# B&R Automation Studio project PickNPlaceD5Demo (part 2)

#### DeviceActions.st
```iecst
ACTION updateProductData:

	FOR i:=0 TO MAX_TRACKING_FRAMES DO
		IF (Products[i].TrackingFrameID <> 0 AND Products[i].Attribute <> 0) THEN
			ProdDetails ACCESS Products[i].Attribute;
			brsmemcpy(ADR(ProdDetails.Pos), ADR(Products[i].CurrentPosition), SIZEOF(McPosType));
			ProdDetails.This := ADR(ProdDetails);
			ProdDetails.TrackingFrameID := Products[i].TrackingFrameID;
		END_IF
	END_FOR

END_ACTION

ACTION deleteOutOfScopeProducts:

	FOR i:=0 TO MAX_TRACKING_FRAMES DO
		IF Products[i].Distance >= ConvSettings.DeletePosition THEN // todo: distance as a constant!
			IF (Products[i].Attribute <> 0) THEN
				brsmemset(Products[i].Attribute, 0, SIZEOF(ProductDetailsType));
			END_IF
			MC_BR_TrackingFrameDelete_0.Mode := mcTRKFRM_DELETE_MOD_FRAME;
			MC_BR_TrackingFrameDelete_0.TrackingFrameID	:= Products[i].TrackingFrameID;
			MC_BR_TrackingFrameDelete_0.Execute	:= TRUE;
			EXIT;
		END_IF
	END_FOR

END_ACTION

ACTION addNewObjects:

	LastProductPosition := MpAxConveyor.Position;

	// Generate a random Y Position --> Here a vision sensor informatin is needed in real systems
	MC_BR_TrackingFrameCreate_0.Parameters.Translation.Y := ConvSettings.YShift;

	// Add attributes memory
	FOR i := 0 TO MAX_TRACKING_FRAMES DO
		IF ProductDetails[i].TrackingFrameID = 0 THEN
			brsmemset(ADR(ProductDetails[i]), 0, SIZEOF(ProductDetailsType));
			MC_BR_TrackingFrameCreate_0.Parameters.Attribute := ADR(ProductDetails[i]);
			EXIT;
		END_IF
	END_FOR

	// Add frame in the buffer
	MC_BR_TrackingFrameCreate_0.Parameters.LatchedPath.Position := LastProductPosition;
	MC_BR_TrackingFrameCreate_0.Execute	:= TRUE;

END_ACTION

ACTION updateSceneViewerPositions:

	FOR i:= 0 TO MAX_TRACKING_FRAMES DO
		ProductsPosition[i].Valid := Products[i].TrackingFrameID <> 0;

		IF Products[i].Attribute <> 0 THEN
			ProdDetails ACCESS Products[i].Attribute;
			IF ProdDetails.InTracking THEN
				ProductsPosition[i].Material := 4; //yellow
			ELSE
				ProductsPosition[i].Material := 1; //red
			END_IF
			ProductsPosition[i].Full := ProdDetails.Used;
			ProductsPosition[i].Empty := NOT ProdDetails.Used;
			ProductsPosition[i].Element1 := ProdDetails.Element1;
			ProductsPosition[i].Element2 := ProdDetails.Element2;
		ELSE
			ProductsPosition[i].Full := FALSE;
			ProductsPosition[i].Empty := FALSE;
			ProductsPosition[i].Element1 := FALSE;
			ProductsPosition[i].Element2 := FALSE;
			ProductsPosition[i].Material := 1;
		END_IF

		ProductsPosition[i].PositionX := LREAL_TO_REAL(Products[i].CurrentPosition.X);
		ProductsPosition[i].PositionY := LREAL_TO_REAL(Products[i].CurrentPosition.Y);
		ProductsPosition[i].PositionZ := LREAL_TO_REAL(Products[i].CurrentPosition.Z);
	END_FOR

END_ACTION

ACTION applyBeltMovement:

	IF AxWithCommandConsideration THEN
		IF NOT MC_MoveAdditive_0.Busy THEN
			MC_MoveAdditive_0.Distance := ConvSettings.IndexingDistance;
			MC_MoveAdditive_0.Velocity := ConvSettings.VelocityProduction;
			MC_MoveAdditive_0.BufferMode := mcABORTING;
			MC_MoveAdditive_0.Execute := TRUE;
		END_IF
	ELSE
		MC_MoveVelocity_0.Velocity := ConvSettings.VelocityProduction;
		MC_MoveVelocity_0.Execute := MC_MoveVelocity_0.InVelocity OR NOT MC_MoveVelocity_0.Busy;
	END_IF

END_ACTION

ACTION resetFUBs:

	IF (MpAxConveyor.Update AND MpAxConveyor.UpdateDone) OR MpAxConveyor.Error THEN
		MpAxConveyor.Update	:= FALSE;
	END_IF

	IF (NOT(MpAxConveyor.MoveActive) AND NOT(MpAxConveyor.CommandBusy)) OR MpAxConveyor.Error THEN
		MpAxConveyor.MoveVelocity := FALSE;
		MpAxConveyor.Update := FALSE;
	END_IF

	IF MpAxConveyor.ErrorReset AND NOT(MpAxConveyor.Error) THEN
		MpAxConveyor.ErrorReset := FALSE;
	END_IF

	IF (MpAxConveyor.Home AND MpAxConveyor.IsHomed) OR MpAxConveyor.Error THEN
		MpAxConveyor.Home := FALSE;
	END_IF

	IF MC_BR_TrackingFrameCreate_0.Done OR MC_BR_TrackingFrameCreate_0.Error THEN
		MC_BR_TrackingFrameCreate_0.Execute	:= FALSE;
	END_IF

	IF MC_BR_TrackingFrameDelete_0.Done OR MC_BR_TrackingFrameDelete_0.Error THEN
		MC_BR_TrackingFrameDelete_0.Execute := FALSE;
	END_IF

	IF MC_MoveVelocity_0.Error OR MC_MoveVelocity_0.CommandAborted OR MC_MoveVelocity_0.Busy THEN
		MC_MoveVelocity_0.Execute := FALSE;
	END_IF

	IF MC_MoveAdditive_0.Error OR MC_MoveAdditive_0.CommandAborted OR MC_MoveAdditive_0.Busy OR MC_MoveAdditive_0.Done THEN
		MC_MoveAdditive_0.Execute := FALSE;
	END_IF

	IF MC_Stop_0.Error OR MC_Stop_0.CommandAborted OR MC_Stop_0.Busy OR MC_Stop_0.Done THEN
		MC_MoveAdditive_0.Execute := FALSE;
	END_IF

	IF MC_BR_TrackingPathReset_0.Busy OR MC_BR_TrackingPathReset_0.Error OR MC_BR_TrackingPathReset_0.Done THEN
		MC_BR_TrackingPathReset_0.Execute := FALSE;
	END_IF

	IF MC_BR_TrackingPathReadInfo_0.Error THEN
		MC_BR_TrackingPathReadInfo_0.Enable := FALSE;
	END_IF

END_ACTION

ACTION initConveyor:

	// Configure Frame Buffer, to get actual pointer to Products --> Check state of Products
	MC_BR_TrackingPathGetFrames_0.Parameters.CoordSystem := mcACS;
	MC_BR_TrackingPathGetFrames_0.Parameters.DataAddress := ADR(Products);
	MC_BR_TrackingPathGetFrames_0.Parameters.GetMode	:= mcTRKPATH_GET_MOD_ALL_FRAMES;
	MC_BR_TrackingPathGetFrames_0.Parameters.InfoMode	:= mcTRKPATH_INFO_MOD_ALL;
	MC_BR_TrackingPathGetFrames_0.Parameters.NumberOfFrames := MAX_TRACKING_FRAMES;
	MC_BR_TrackingPathGetFrames_0.Parameters.TrackingFrameID := 0;

	// Set Default Parameters of the Tracking Frames
	MC_BR_TrackingFrameCreate_0.Parameters.Attribute	:= 0;
	MC_BR_TrackingFrameCreate_0.Parameters.Translation.X := 0.0;
	MC_BR_TrackingFrameCreate_0.Parameters.Translation.Y := 0.0;
	MC_BR_TrackingFrameCreate_0.Parameters.Translation.Z := 0.0;
	MC_BR_TrackingFrameCreate_0.Parameters.Orientation.Angle1 := 0.0;
	MC_BR_TrackingFrameCreate_0.Parameters.Orientation.Angle2 := 0.0;
	MC_BR_TrackingFrameCreate_0.Parameters.Orientation.Angle3 := 0.0;
	MC_BR_TrackingFrameCreate_0.Parameters.Orientation.Type := 0;

	MC_BR_TrackingPathReadStatus_0.Enable := TRUE;
	MC_BR_TrackingPathReadInfo_0.Enable := TRUE;

	// Configuration of movement command
	MC_MoveAdditive_0.Acceleration := 1000;
	MC_MoveAdditive_0.Deceleration := 1000;
	MC_MoveAdditive_0.Jerk := 10000;
	MC_MoveAdditive_0.BufferMode := mcABORTING;

	MC_MoveVelocity_0.Acceleration := 1000;
	MC_MoveVelocity_0.Deceleration := 1000;
	MC_MoveVelocity_0.Direction := mcDIR_POSITIVE;
	MC_MoveVelocity_0.BufferMode := mcABORTING;

	MC_Stop_0.Deceleration := 1000;
	MC_Stop_0.Jerk := 10000;

	// Belt Position of fixed tracking frame
	ParkPosition := 0;

END_ACTION
```

### Program Logical/Conveyor/APP_ConveyorOut (IEC)

#### Init.st
```iecst
PROGRAM _INIT

	TrackLinkConveyor := ADR(gTrackingPathConveyorOut);
	AxGroupLink := ADR(AxConveyorOut);
	ConvSettings ACCESS ADR(ControlPanel.Input.Conveyor2);
	AxWithCommandConsideration := TRUE;

	initConveyor;

END_PROGRAM
```

- Cyclic.st (reference to Logical/Conveyor/APP_ConveyorIn/Cyclic.st)

- DeviceActions.st (reference to Logical/Conveyor/APP_ConveyorIn/DeviceActions.st)

- Variables.var (reference to Logical/Conveyor/APP_ConveyorIn/Variables.var)

### Package Logical/Robots/Robot1 - Device: Scara

### Program Logical/Robots/Robot1/APP_Robot1

#### CommonVars.var
```iecst
(*
Link handling*)
VAR
	AxQ1 : UDINT; (*Memory to Q1*)
	AxQ2 : UDINT; (*Memory to Q2*)
	AxQ3 : UDINT; (*Memory to Q4*)
	AxQ4 : UDINT; (*Memory to Q4*)
	AxQ5 : UDINT; (*Memory to Q4*)
	TrackLinkConveyorOut : UDINT; (*Link to conveyor tracking path*)
	TrackLinkConveyorIn : UDINT; (*Link to conveyor tracking path*)
	MpDeltaName : STRING[250]; (*Name of axGroup to find position in object hierachy*)
	MpLinkDelta : UDINT; (*Link to delta*)
	ProgramLink : REFERENCE TO STRING[32]; (*Program name as string executed by the interpreter*)
END_VAR
(*
Robot Definition*)
VAR
	MC_BR_MoveProgram_X : MC_BR_MoveProgram;
	MC_BR_GroupPower_X : MC_BR_GroupPower;
	MC_GroupStop_X : MC_GroupStop;
	MC_GroupReset_X : MC_GroupReset;
	MC_BR_GroupHome_X : MC_BR_GroupHome_15; (*Group object to home axis group*)
	MC_BR_GroupReadInfo_X : MC_BR_GroupReadInfo;
	MC_GroupContinue_X : MC_GroupContinue; (*Continue Interpreter in case of a new tracking Object*)
	MC_BR_TrackingStatus_PathGen_X : MC_BR_TrackingStatus_PathGen; (*Tracking Path, read all objects on Path*)
	MC_BR_PathInfo_X : MC_BR_PathInfo;
	MC_GroupReadStatus_X : MC_GroupReadStatus; (*Group object to home axis group*)
	MC_BR_PauseWorkspaceMonitoring_X : MC_BR_PauseWorkspaceMonitoring;
	MC_GroupReadActualPosition_X : MC_GroupReadActualPosition_15; (*Group object to home axis group*)
END_VAR
(*
Variables used handling objects and reading informations about the robot*)
VAR
	MC_BR_TrackingPathGetFrames_In : MC_BR_TrackingPathGetFrames; (*Tracking Path, read all objects on Path*)
	MC_BR_TrackingPathReadStatus_In : MC_BR_TrackingPathReadStatus;
	MC_BR_TrackingPathGetFrames_Out : MC_BR_TrackingPathGetFrames; (*Tracking Path, read all objects on Path*)
	MC_BR_TrackingPathReadStatus_Out : MC_BR_TrackingPathReadStatus;
END_VAR
(*
Logic*)
VAR
	State : DeviceStatesListEnum; (*Statemachine*)
	i : INT; (*loop counter*)
	j : INT; (*loop counter*)
	XPosMax : LREAL; (*Figure out object with min distance to the robot*)
	FeedrateReduction : LREAL; (*Feedrate reduction calculated based on the distance*)
	Products_Out : ARRAY[0..MAX_TRACKING_FRAMES] OF McTrkFrmInfoType; (*List of all Frames*)
	Products_In : ARRAY[0..MAX_TRACKING_FRAMES] OF McTrkFrmInfoType; (*List of all Frames*)
END_VAR
(*
Scene Viewer*)
VAR
	ProdDetails : REFERENCE TO ProductDetailsType; (*Scene Viewer*)
	PickTrackingObjectDetails : REFERENCE TO ProductDetailsType; (*Scene Viewer*)
	PlaceTrackingObjectDetails : REFERENCE TO ProductDetailsType; (*Scene Viewer*)
	Grab1Closed : BOOL;
	Grab2Closed : BOOL;
END_VAR
(*
ST Var*)
VAR
	MinPlacePosX : LREAL := 0; (*ST Var - Maximum reachable x position*)
	MaxPlacePosX : LREAL := 0; (*ST Var - Maximum reachable x position*)
	MinPickPosX : LREAL := 0; (*ST Var - Maximum reachable x position*)
	MaxPickPosX : LREAL := 0; (*ST Var - Maximum reachable x position*)
	PlaceTrackingObject : UDINT; (*ST Var - ADR(ProductDetailsType)*)
	PickTrackingObject : UDINT; (*ST Var - ADR(ProductDetailsType)*)
	M8 : BOOL; (*ST Var*)
	M9 : BOOL; (*ST Var*)
	M16 : BOOL; (*ST Var*)
	M17 : BOOL; (*ST Var*)
	M20 : BOOL; (*ST Var*)
	M21 : BOOL; (*ST Var*)
END_VAR
(*
Monitorin Elements*)
VAR
	BasicMonitor : McPathGenMonElemBasicMonType; (*Monitor to get interpreter line*)
	IPMonitor : McProgIntIpMonitorType; (*Monitor to get interpreter line*)
END_VAR
```

#### Cyclic.st
```iecst
PROGRAM _CYCLIC

	CASE State OF

		/////////////////////////////////////////////////////////////////////////////
		STATE_WAIT:
		/////////////////////////////////////////////////////////////////////////////
			IF  ControlPanel.Input.Start THEN
				State := STATE_INIT;
			END_IF

		/////////////////////////////////////////////////////////////////////////////
		STATE_INIT:
			/////////////////////////////////////////////////////////////////////////////
			IF NOT (MC_BR_TrackingPathReadStatus_In.TrackingPathReady OR MC_BR_TrackingPathReadStatus_Out.TrackingPathReady) THEN
				/// Wait
			ELSIF MC_BR_GroupHome_X.Busy OR MC_GroupReset_X.Busy OR NOT MC_GroupReadStatus_X.Valid OR NOT MC_BR_GroupReadInfo_X.Valid THEN
				// wait
			ELSIF MC_GroupReadStatus_X.Error OR MC_BR_GroupHome_X.Error OR MC_BR_GroupPower_X.Error OR MC_BR_MoveProgram_X.Error OR MC_GroupReset_X.Error OR MC_BR_GroupReadInfo_X.Error THEN
				MC_GroupReset_X.Execute := TRUE;

			ELSIF NOT MC_BR_GroupReadInfo_X.PowerOn THEN
				MC_BR_GroupPower_X.Enable := TRUE;

			ELSIF NOT MC_BR_GroupReadInfo_X.IsHomed	THEN
				MC_BR_GroupHome_X.Execute := TRUE;

			ELSIF MC_GroupReadStatus_X.GroupStandby THEN
				PickTrackingObject := 0;
				PlaceTrackingObject := 0;
				brsmemset(ADR(Products_In), 0, SIZEOF(Products_In));
				brsmemset(ADR(Products_Out), 0, SIZEOF(Products_Out));
				MC_BR_MoveProgram_X.Name := ProgramLink;
				MC_BR_MoveProgram_X.Execute := TRUE;
				MC_BR_PauseWorkspaceMonitoring_X.Enable := FALSE;
				State := STATE_PRODUCTION;

			END_IF

		/////////////////////////////////////////////////////////////////////////////
		STATE_PRODUCTION:
		/////////////////////////////////////////////////////////////////////////////

			// ------------------------------------------------------------------------------------------------------------------------------------------------
			// Case Pick Frame: choose which frame is the next to pick which is not already grabbed and not already in manipulation
			// ------------------------------------------------------------------------------------------------------------------------------------------------
			chooseNextSlots;

			// ------------------------------------------------------------------------------------------------------------------------------------------------
			// Case Grip Product: Hande M Commands on Tracked object
			// ------------------------------------------------------------------------------------------------------------------------------------------------
			handleMFunctions;

			// ------------------------------------------------------------------------------------------------------------------------------------------------
			// Case Scene Viewer Update Robot 1: Update Positions in Tracking case, to get a Scene Viewer Visu
			// ------------------------------------------------------------------------------------------------------------------------------------------------

			updateSceneViewer;

			// ------------------------------------------------------------------------------------------------------------------------------------------------
			// Case State M. Production : Handle End of Process
			// ------------------------------------------------------------------------------------------------------------------------------------------------
			IF MC_GroupReadStatus_X.Error OR MC_GroupReadStatus_X.GroupErrorStop OR MC_BR_MoveProgram_X.Error THEN
				State := STATE_ERROR;
				MC_GroupStop_X.Execute := TRUE;
				ControlPanel.Input.Start := FALSE;

			ELSIF NOT(ControlPanel.Input.Start) THEN

				MC_GroupStop_X.Execute := TRUE;
				MC_BR_GroupPower_X.Enable := FALSE;

				IF MC_GroupReadStatus_X.GroupDisabled THEN
					State := STATE_WAIT;

				ELSIF MC_GroupReadStatus_X.GroupErrorStop THEN
					State := STATE_ERROR;
				END_IF

			END_IF

		///////////////////////////////////////////////////////////////////////////////
		STATE_ERROR:
		///////////////////////////////////////////////////////////////////////////////
			IF MC_GroupReset_X.Busy OR MC_GroupReadStatus_X.Error OR MC_GroupReadStatus_X.GroupErrorStop THEN
				IF ControlPanel.Input.Reset THEN
					MC_GroupReset_X.Execute := NOT MC_GroupReset_X.Busy;
					MC_BR_GroupHome_X.Execute := NOT MC_BR_GroupHome_X.Busy;
				END_IF
			ELSE
				State := STATE_WAIT;
			END_IF

	END_CASE

	PlaceTrackingObjectDetails ACCESS PlaceTrackingObject;
	PickTrackingObjectDetails ACCESS PickTrackingObject;
	runFUBs;

END_PROGRAM
```

#### DefineLinks.st
```iecst
ACTION DefineLinks:

	// Define Links to the axes of the Robot
	AxQ1 := ADR(gAxisQ1_D5r1100R_1);
	AxQ2 := ADR(gAxisQ2_D5r1100R_1);
	AxQ3 := ADR(gAxisQ3_D5r1100R_1);
	AxQ4 := ADR(gAxisQ4_D5r1100R_1);
	AxQ5 := ADR(gAxisQ5_D5r1100R_1);

	// Define Link to the Robot & Conveyor
	MpDeltaName	:= 'gAxesGroup_D5r1100R_1';
	MpLinkDelta	:= ADR(gAxesGroup_D5r1100R_1);
	TrackLinkConveyorIn := ADR(gTrackingPathConveyorIn);
	TrackLinkConveyorOut := ADR(gTrackingPathConveyorOut);

	// Define Link to Interpreter Program
	ProgramLink ACCESS ADR(ControlPanel.Input.ProgramRobot1);

END_ACTION
```

#### DeviceActions.st
```iecst
// This action choses the next Product to be manipulated by the robot
ACTION chooseNextSlots:
	XPosMax := 0;
	j := MAX_TRACKING_FRAMES + 1;
	FOR i := 0 TO MAX_TRACKING_FRAMES DO
		IF Products_In[i].TrackingFrameID <> 0 AND
			Products_In[i].Attribute <> 0 AND
			Products_In[i].TrackingFrameID <> MC_BR_TrackingStatus_PathGen_X.TrackingAdditionalInfo.TrackedFrame.FrameId THEN
			ProdDetails ACCESS Products_In[i].Attribute;

			// current frame is suitable - find the optimal one
			IF ProdDetails.Used = FALSE  AND	// no other robot has manipulate this object
				Products_In[i].Distance < (MaxPickPosX) AND // not already outside of the position
				Products_In[i].Distance > XPosMax AND // the object is the nearest to the robot
				Products_In[i].Distance > (MinPickPosX) THEN // product is within the scope of the robot
				// select as next object
				XPosMax := Products_In[i].Distance;
				j := i;
			END_IF
		END_IF
	END_FOR

	IF j <= MAX_TRACKING_FRAMES THEN
		PickTrackingObject := Products_In[j].Attribute;
		MC_GroupContinue_X.Execute := MC_BR_GroupReadInfo_X.AdditionalInfo.GroupInterrupted AND NOT MC_GroupContinue_X.Busy ;
	ELSE
		PickTrackingObject := 0;
	END_IF

	XPosMax := 0;
	j := MAX_TRACKING_FRAMES + 1;
	FOR i := 0 TO MAX_TRACKING_FRAMES DO
		IF Products_Out[i].TrackingFrameID <> 0 AND
			Products_Out[i].Attribute <> 0 AND
			Products_Out[i].TrackingFrameID <> MC_BR_TrackingStatus_PathGen_X.TrackingAdditionalInfo.TrackedFrame.FrameId THEN
			ProdDetails ACCESS Products_Out[i].Attribute;

			// current frame is suitable - find the optimal one
			IF ProdDetails.Used = FALSE  AND	// no other robot has manipulate this object
				Products_Out[i].Distance < (MaxPlacePosX) AND // not already outside of the position
				Products_Out[i].Distance > XPosMax AND // the object is the nearest to the robot
				Products_Out[i].Distance > (MinPlacePosX) THEN // product is within the scope of the robot
				// select as next object
				XPosMax := Products_Out[i].Distance;
				j := i;
			END_IF
		END_IF
	END_FOR

	IF j <= MAX_TRACKING_FRAMES THEN
		PlaceTrackingObject := Products_Out[j].Attribute;
	ELSE
		PlaceTrackingObject := 0;
	END_IF

END_ACTION

// This action operates the Gripper,
ACTION handleMFunctions:
	FOR i := 0 TO MAX_TRACKING_FRAMES DO
		IF MC_BR_TrackingStatus_PathGen_X.TrackingAdditionalInfo.TrackedFrame.FrameId <> 0 THEN
			ProdDetails ACCESS 0;
			IF MC_BR_TrackingStatus_PathGen_X.TrackingAdditionalInfo.TrackedFrame.FrameId = Products_In[i].TrackingFrameID THEN
				ProdDetails ACCESS Products_In[i].Attribute;
			END_IF
			IF MC_BR_TrackingStatus_PathGen_X.TrackingAdditionalInfo.TrackedFrame.FrameId = Products_Out[i].TrackingFrameID THEN
				ProdDetails ACCESS Products_Out[i].Attribute;
			END_IF

			IF ADR(ProdDetails) <> 0 THEN
				IF M8 OR M9 OR M16 OR M17 THEN
					ProdDetails.Used := TRUE;
				END_IF

				IF M8 THEN
					ProdDetails.Element1 := FALSE;
				END_IF

				IF M9 THEN
					ProdDetails.Element2 := FALSE;
				END_IF

				IF M16 THEN
					ProdDetails.Element1 := TRUE;
				END_IF

				IF M17 THEN
					ProdDetails.Element2 := TRUE;
				END_IF

			END_IF
		END_IF
	END_FOR

	IF M8 THEN
		Grab1Closed := TRUE;
	END_IF

	IF M16 THEN
		Grab1Closed := FALSE;
	END_IF

	IF M9 THEN
		Grab2Closed := TRUE;
	END_IF

	IF M17 THEN
		Grab2Closed := FALSE;
	END_IF

	IF M20 THEN
		MC_BR_PauseWorkspaceMonitoring_X.Enable := TRUE;
	END_IF

	IF M21 THEN
		MC_BR_PauseWorkspaceMonitoring_X.Enable := FALSE;
	END_IF

	M8 := FALSE;
	M16 := FALSE;
	M9 := FALSE;
	M17 := FALSE;
	M20 := FALSE;
	M21 := FALSE;
END_ACTION

ACTION runFUBs:

	MC_BR_GroupHome_X(AxesGroup := MpLinkDelta);
	MC_GroupStop_X(AxesGroup := MpLinkDelta);
	MC_BR_MoveProgram_X(AxesGroup := MpLinkDelta);
	MC_BR_GroupPower_X(AxesGroup := MpLinkDelta);
	MC_GroupReset_X(AxesGroup := MpLinkDelta);
	MC_GroupReadStatus_X(AxesGroup := MpLinkDelta);
	MC_BR_GroupReadInfo_X(AxesGroup := MpLinkDelta);
	MC_BR_TrackingStatus_PathGen_X(AxesGroup := MpLinkDelta);
	MC_BR_PathInfo_X(AxesGroup := MpLinkDelta);
	MC_GroupContinue_X(AxesGroup := MpLinkDelta);
	MC_GroupReadActualPosition_X(AxesGroup := MpLinkDelta);
	MC_BR_PauseWorkspaceMonitoring_X(AxesGroup := MpLinkDelta);

	MC_GroupReset_X.Execute := MC_GroupReset_X.Execute AND NOT (MC_GroupReset_X.Done OR MC_GroupReset_X.Error);
	MC_GroupStop_X.Execute := MC_GroupStop_X.Execute AND NOT (MC_GroupStop_X.Done OR MC_GroupStop_X.Error OR MC_GroupStop_X.CommandAborted);
	MC_BR_MoveProgram_X.Execute := MC_BR_MoveProgram_X.Execute AND NOT (MC_BR_MoveProgram_X.Done OR MC_BR_MoveProgram_X.Error OR MC_BR_MoveProgram_X.CommandAborted);
	MC_BR_GroupHome_X.Execute := MC_BR_GroupHome_X.Execute AND NOT (MC_BR_GroupHome_X.Done OR MC_BR_GroupHome_X.Error OR MC_BR_GroupHome_X.CommandAborted);
	MC_BR_GroupPower_X.Enable := MC_BR_GroupPower_X.Enable AND NOT (MC_BR_GroupPower_X.Error);
	MC_GroupContinue_X.Execute := MC_GroupContinue_X.Execute AND NOT (MC_GroupContinue_X.Done OR MC_GroupContinue_X.Error OR MC_GroupContinue_X.CommandAborted);

	// Tracking of moving objects
	MC_BR_TrackingPathReadStatus_In();
	MC_BR_TrackingPathGetFrames_In();
	MC_BR_TrackingPathReadStatus_Out();
	MC_BR_TrackingPathGetFrames_Out();

	// Toogle Execution - needed cause FUB detects positive edge
	IF MC_BR_TrackingPathReadStatus_In.TrackingPathErrorStop OR MC_BR_TrackingPathReadStatus_In.TrackingPathErrorStop THEN
		brsmemset(ADR(Products_Out), 0, SIZEOF(Products_Out));
		brsmemset(ADR(Products_In), 0, SIZEOF(Products_In));
		MC_BR_TrackingPathGetFrames_In.Execute := FALSE;
		MC_BR_TrackingPathGetFrames_Out.Execute := FALSE;
	ELSE
		MC_BR_TrackingPathGetFrames_In.Execute := NOT(MC_BR_TrackingPathGetFrames_In.Done) AND NOT (MC_BR_TrackingPathGetFrames_In.Error);
		MC_BR_TrackingPathGetFrames_Out.Execute := NOT(MC_BR_TrackingPathGetFrames_Out.Done) AND NOT (MC_BR_TrackingPathGetFrames_Out.Error);
	END_IF

	IF NOT IPMonitor.Handshake THEN
		IPMonitor.Handshake := TRUE;
	END_IF

END_ACTION

ACTION updateSceneViewer:

	// ------------------------------------------------------------------------------------------------------------------------------------------------
	// Highliting of actual object tracked for Scene Viewer visu
	// ------------------------------------------------------------------------------------------------------------------------------------------------

	FOR i := 0 TO MAX_TRACKING_FRAMES DO
		IF Products_In[i].Attribute <> 0 THEN
			ProdDetails ACCESS Products_In[i].Attribute;
			IF MC_BR_TrackingStatus_PathGen_X.TrackingAdditionalInfo.TrackedFrame.FrameId = ProdDetails.TrackingFrameID AND
				MC_BR_TrackingStatus_PathGen_X.TrackingAdditionalInfo.TrackedFrame.FrameId <> 0 THEN
				ProdDetails.InTracking := TRUE;
			ELSE
				ProdDetails.InTracking := FALSE;
			END_IF
		END_IF
	END_FOR

	FOR i := 0 TO MAX_TRACKING_FRAMES DO
		IF Products_Out[i].Attribute <> 0 THEN
			ProdDetails ACCESS Products_Out[i].Attribute;
			IF MC_BR_TrackingStatus_PathGen_X.TrackingAdditionalInfo.TrackedFrame.FrameId = ProdDetails.TrackingFrameID AND
				MC_BR_TrackingStatus_PathGen_X.TrackingAdditionalInfo.TrackedFrame.FrameId <> 0 THEN
				ProdDetails.InTracking := TRUE;
			ELSE
				ProdDetails.InTracking := FALSE;
			END_IF
		END_IF
	END_FOR

END_ACTION
```

#### Init.st
```iecst
PROGRAM _INIT

	// This action defines the links to the conveyeor and the robot
	DefineLinks;

	// M-Functions triggered in Interpreter Program
	M8;
	M9;
	M16;
	M17;

	MC_BR_TrackingPathReadStatus_In.TrackingPath 				:= TrackLinkConveyorIn;
	MC_BR_TrackingPathReadStatus_In.Enable						:= TRUE;
	MC_BR_TrackingPathGetFrames_In.TrackingPath 				:= TrackLinkConveyorIn;
	MC_BR_TrackingPathGetFrames_In.Parameters.CoordSystem		:= mcACS;
	MC_BR_TrackingPathGetFrames_In.Parameters.DataAddress 		:= ADR(Products_In);
	MC_BR_TrackingPathGetFrames_In.Parameters.GetMode			:= mcTRKPATH_GET_MOD_ALL_FRAMES;
	MC_BR_TrackingPathGetFrames_In.Parameters.InfoMode			:= mcTRKPATH_INFO_MOD_ALL;
	MC_BR_TrackingPathGetFrames_In.Parameters.NumberOfFrames 	:= SIZEOF(Products_In)/SIZEOF(McTrkFrmInfoType);
	MC_BR_TrackingPathGetFrames_In.Parameters.TrackingFrameID 	:= 0;

	MC_BR_TrackingPathReadStatus_Out.TrackingPath 				:= TrackLinkConveyorOut;
	MC_BR_TrackingPathReadStatus_Out.Enable						:= TRUE;
	MC_BR_TrackingPathGetFrames_Out.TrackingPath 				:= TrackLinkConveyorOut;
	MC_BR_TrackingPathGetFrames_Out.Parameters.CoordSystem		:= mcACS;
	MC_BR_TrackingPathGetFrames_Out.Parameters.DataAddress 		:= ADR(Products_Out);
	MC_BR_TrackingPathGetFrames_Out.Parameters.GetMode			:= mcTRKPATH_GET_MOD_ALL_FRAMES;
	MC_BR_TrackingPathGetFrames_Out.Parameters.InfoMode			:= mcTRKPATH_INFO_MOD_ALL;
	MC_BR_TrackingPathGetFrames_Out.Parameters.NumberOfFrames 	:= SIZEOF(Products_Out)/SIZEOF(McTrkFrmInfoType);
	MC_BR_TrackingPathGetFrames_Out.Parameters.TrackingFrameID 	:= 0;

	MC_GroupReadActualPosition_X.CoordSystem := mcMCS;
	MC_GroupReadActualPosition_X.Enable := TRUE;

	// Offset of the Robot (Object Hierachy)
	MC_BR_TrackingStatus_PathGen_X.Enable := TRUE;
	MC_BR_GroupReadInfo_X.Enable := TRUE;
	MC_GroupReadStatus_X.Enable := TRUE;
	MC_BR_PathInfo_X.Enable := TRUE;

END_PROGRAM
```

Listed in the project but not available here: FileDevices/GCode/ProdDetails.typ, Logical/GeneralTexts, Logical/Conveyor/APP_ConveyorIn/Exit.st, Logical/Conveyor/APP_ConveyorIn/Exit.st, Logical/Scene3D
